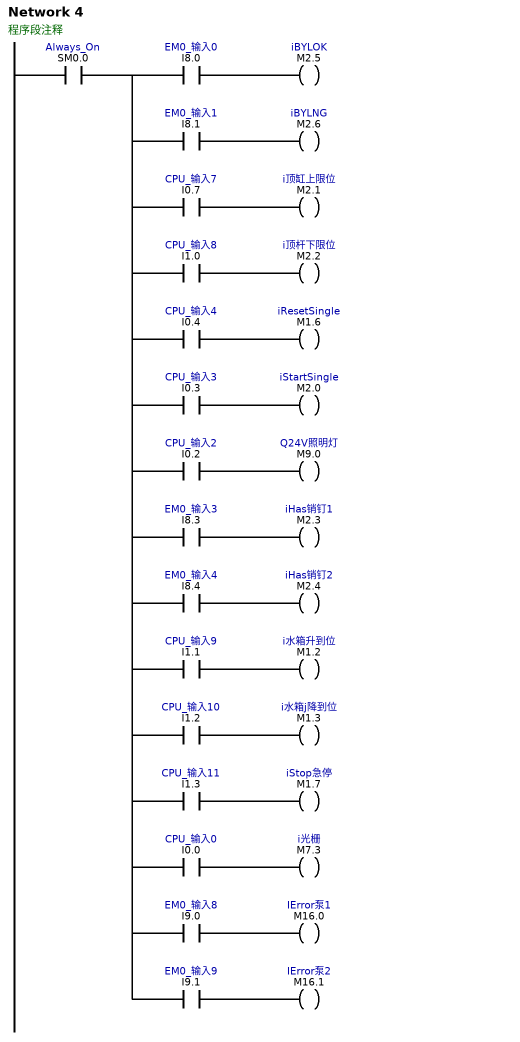
[picture p24: SBR5 networks 4-4]
Network 4
// 程序段注释
LD     Always_On:SM0.0
LPS
A      EM0_输入0:I8.0
=      iBYLOK:M2.5
LRD
A      EM0_输入1:I8.1
=      iBYLNG:M2.6
LRD
A      CPU_输入7:I0.7
=      i顶缸上限位:M2.1
LRD
A      CPU_输入8:I1.0
=      i顶杆下限位:M2.2
LRD
A      CPU_输入4:I0.4
=      iResetSingle:M1.6
LRD
A      CPU_输入3:I0.3
=      iStartSingle:M2.0
LRD
A      CPU_输入2:I0.2
=      Q24V照明灯:M9.0
LRD
A      EM0_输入3:I8.3
=      iHas销钉1:M2.3
LRD
A      EM0_输入4:I8.4
=      iHas销钉2:M2.4
LRD
A      CPU_输入9:I1.1
=      i水箱升到位:M1.2
LRD
A      CPU_输入10:I1.2
=      i水箱j降到位:M1.3
LRD
A      CPU_输入11:I1.3
=      iStop急停:M1.7
LRD
A      CPU_输入0:I0.0
=      i光栅:M7.3
LRD
A      EM0_输入8:I9.0
=      IError泵1:M16.0
LPP
A      EM0_输入9:I9.1
=      IError泵2:M16.1
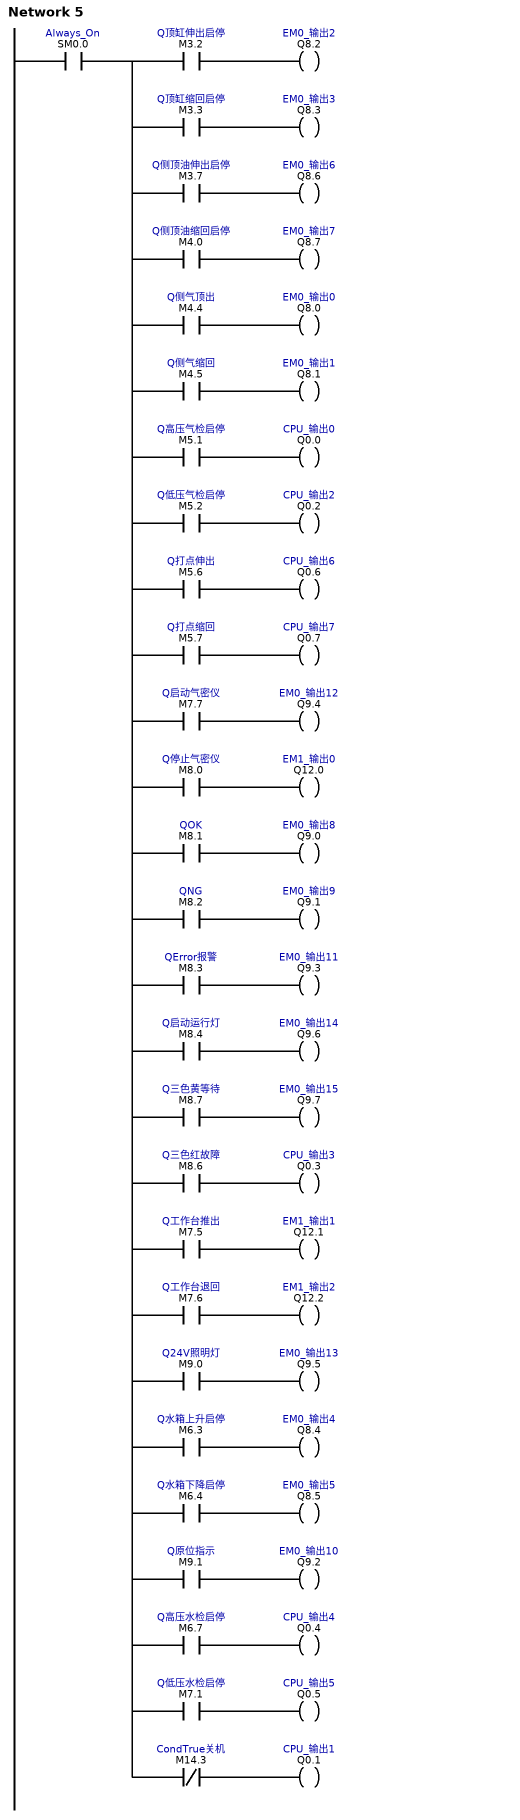
Network 5
LD     Always_On:SM0.0
LPS
A      Q顶缸伸出启停:M3.2
=      EM0_输出2:Q8.2
LRD
A      Q顶缸缩回启停:M3.3
=      EM0_输出3:Q8.3
LRD
A      Q侧顶油伸出启停:M3.7
=      EM0_输出6:Q8.6
LRD
A      Q侧顶油缩回启停:M4.0
=      EM0_输出7:Q8.7
LRD
A      Q侧气顶出:M4.4
=      EM0_输出0:Q8.0
LRD
A      Q侧气缩回:M4.5
=      EM0_输出1:Q8.1
LRD
A      Q高压气检启停:M5.1
=      CPU_输出0:Q0.0
LRD
A      Q低压气检启停:M5.2
=      CPU_输出2:Q0.2
LRD
A      Q打点伸出:M5.6
=      CPU_输出6:Q0.6
LRD
A      Q打点缩回:M5.7
=      CPU_输出7:Q0.7
LRD
A      Q启动气密仪:M7.7
=      EM0_输出12:Q9.4
LRD
A      Q停止气密仪:M8.0
=      EM1_输出0:Q12.0
LRD
A      QOK:M8.1
=      EM0_输出8:Q9.0
LRD
A      QNG:M8.2
=      EM0_输出9:Q9.1
LRD
A      QError报警:M8.3
=      EM0_输出11:Q9.3
LRD
A      Q启动运行灯:M8.4
=      EM0_输出14:Q9.6
LRD
A      Q三色黄等待:M8.7
=      EM0_输出15:Q9.7
LRD
A      Q三色红故障:M8.6
=      CPU_输出3:Q0.3
LRD
A      Q工作台推出:M7.5
=      EM1_输出1:Q12.1
LRD
A      Q工作台退回:M7.6
=      EM1_输出2:Q12.2
LRD
A      Q24V照明灯:M9.0
=      EM0_输出13:Q9.5
LRD
A      Q水箱上升启停:M6.3
=      EM0_输出4:Q8.4
LRD
A      Q水箱下降启停:M6.4
=      EM0_输出5:Q8.5
LRD
A      Q原位指示:M9.1
=      EM0_输出10:Q9.2
LRD
A      Q高压水检启停:M6.7
=      CPU_输出4:Q0.4
LRD
A      Q低压水检启停:M7.1
=      CPU_输出5:Q0.5
LPP
AN     CondTrue关机:M14.3
=      CPU_输出1:Q0.1
END_SUBROUTINE_BLOCK

SUBROUTINE_BLOCK ConverData:SBR6
TITLE=子程序注释
VAR
tmpDint:DINT;	// LD0 
tmpReal:REAL;	// LD4 
END_VAR
BEGIN
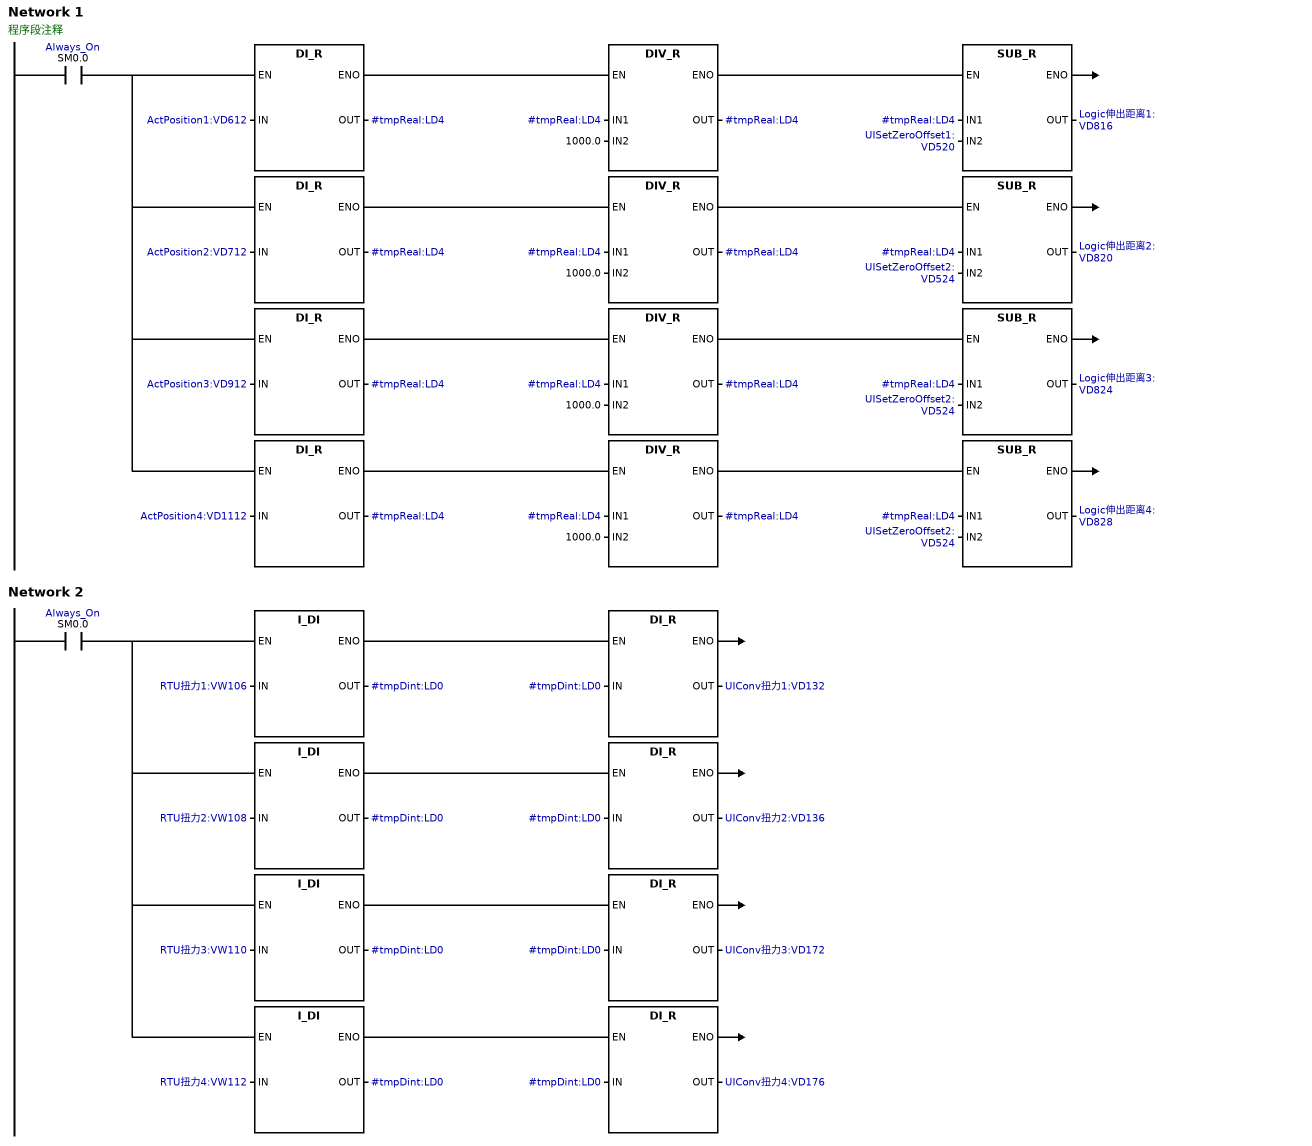
Network 1
// 程序段注释
LD     Always_On:SM0.0
LPS
DTR    ActPosition1:VD612, #tmpReal:LD4
AENO
/R     1000.0, #tmpReal:LD4
AENO
MOVR   #tmpReal:LD4, Logic伸出距离1:VD816
-R     UISetZeroOffset1:VD520, Logic伸出距离1:VD816
LRD
DTR    ActPosition2:VD712, #tmpReal:LD4
AENO
/R     1000.0, #tmpReal:LD4
AENO
MOVR   #tmpReal:LD4, Logic伸出距离2:VD820
-R     UISetZeroOffset2:VD524, Logic伸出距离2:VD820
LRD
DTR    ActPosition3:VD912, #tmpReal:LD4
AENO
/R     1000.0, #tmpReal:LD4
AENO
MOVR   #tmpReal:LD4, Logic伸出距离3:VD824
-R     UISetZeroOffset2:VD524, Logic伸出距离3:VD824
LPP
DTR    ActPosition4:VD1112, #tmpReal:LD4
AENO
/R     1000.0, #tmpReal:LD4
AENO
MOVR   #tmpReal:LD4, Logic伸出距离4:VD828
-R     UISetZeroOffset2:VD524, Logic伸出距离4:VD828
Network 2
LD     Always_On:SM0.0
LPS
ITD    RTU扭力1:VW106, #tmpDint:LD0
AENO
DTR    #tmpDint:LD0, UIConv扭力1:VD132
LRD
ITD    RTU扭力2:VW108, #tmpDint:LD0
AENO
DTR    #tmpDint:LD0, UIConv扭力2:VD136
LRD
ITD    RTU扭力3:VW110, #tmpDint:LD0
AENO
DTR    #tmpDint:LD0, UIConv扭力3:VD172
LPP
ITD    RTU扭力4:VW112, #tmpDint:LD0
AENO
DTR    #tmpDint:LD0, UIConv扭力4:VD176
END_SUBROUTINE_BLOCK

// SBR7: protected block, not included

// SBR8: protected block, not included

SUBROUTINE_BLOCK XinJiePN:SBR9
TITLE=子程序注释
VAR
tmpSpeed:DWORD;	// LD0 
tmpPos1:DINT;	// LD4 
tmpWarning:WORD;	// LW8 
tmpErr:WORD;	// LW10 
tmpDone:BOOL;	// L12.0 
tmpNotJOD:BOOL;	// L12.1 
tmpPos2:DINT;	// LD13 
tmpReal:REAL;	// LD17 
tmpDint:DINT;	// LD21 
tmpPos3:DINT;	// LD25 
tmpPos4:DINT;	// LD29 
END_VAR
BEGIN
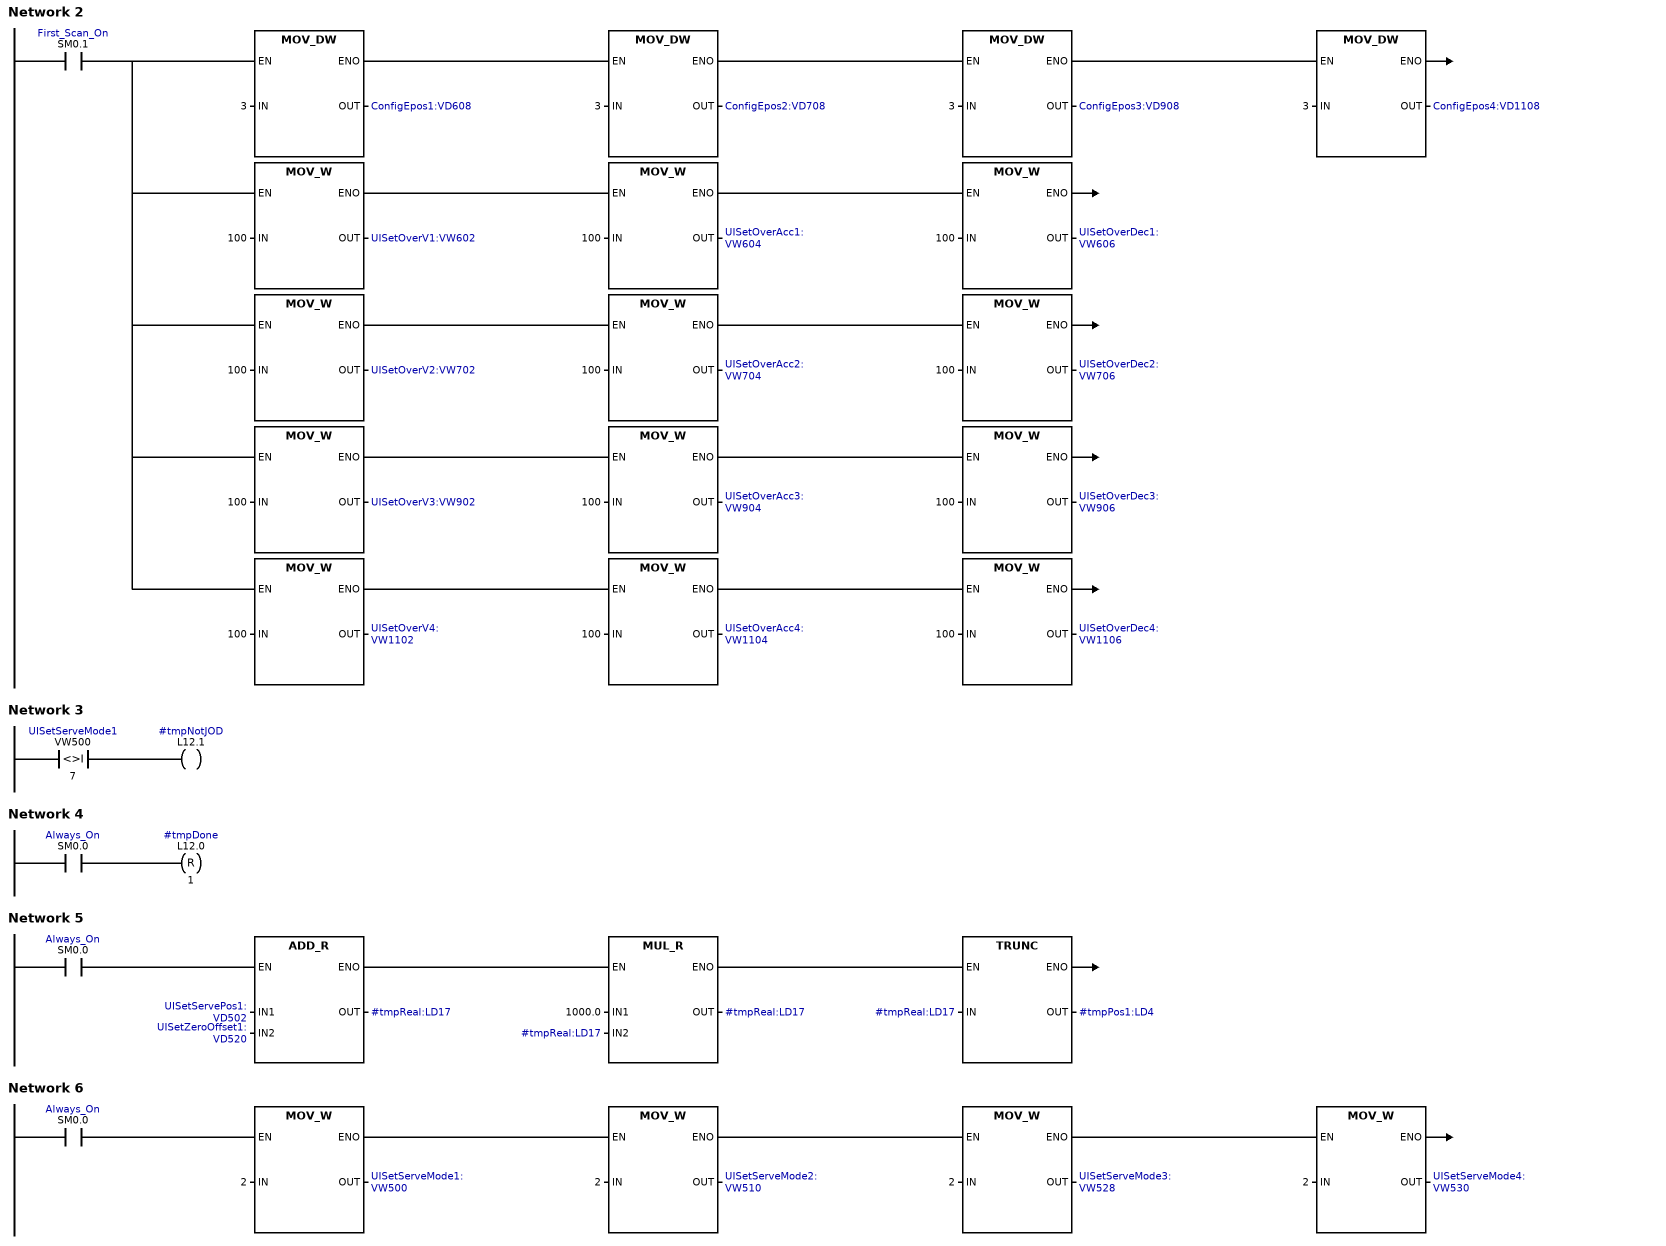
Network 2
LD     First_Scan_On:SM0.1
LPS
MOVD   3, ConfigEpos1:VD608
AENO
MOVD   3, ConfigEpos2:VD708
AENO
MOVD   3, ConfigEpos3:VD908
AENO
MOVD   3, ConfigEpos4:VD1108
LRD
MOVW   100, UISetOverV1:VW602
AENO
MOVW   100, UISetOverAcc1:VW604
AENO
MOVW   100, UISetOverDec1:VW606
LRD
MOVW   100, UISetOverV2:VW702
AENO
MOVW   100, UISetOverAcc2:VW704
AENO
MOVW   100, UISetOverDec2:VW706
LRD
MOVW   100, UISetOverV3:VW902
AENO
MOVW   100, UISetOverAcc3:VW904
AENO
MOVW   100, UISetOverDec3:VW906
LPP
MOVW   100, UISetOverV4:VW1102
AENO
MOVW   100, UISetOverAcc4:VW1104
AENO
MOVW   100, UISetOverDec4:VW1106
Network 3
LDW<>  UISetServeMode1:VW500, 7
=      #tmpNotJOD:L12.1
Network 4
LD     Always_On:SM0.0
R      #tmpDone:L12.0, 1
Network 5
LD     Always_On:SM0.0
MOVR   UISetServePos1:VD502, #tmpReal:LD17
AENO
+R     UISetZeroOffset1:VD520, #tmpReal:LD17
AENO
*R     1000.0, #tmpReal:LD17
AENO
TRUNC  #tmpReal:LD17, #tmpPos1:LD4
Network 6
LD     Always_On:SM0.0
MOVW   2, UISetServeMode1:VW500
AENO
MOVW   2, UISetServeMode2:VW510
AENO
MOVW   2, UISetServeMode3:VW528
AENO
MOVW   2, UISetServeMode4:VW530
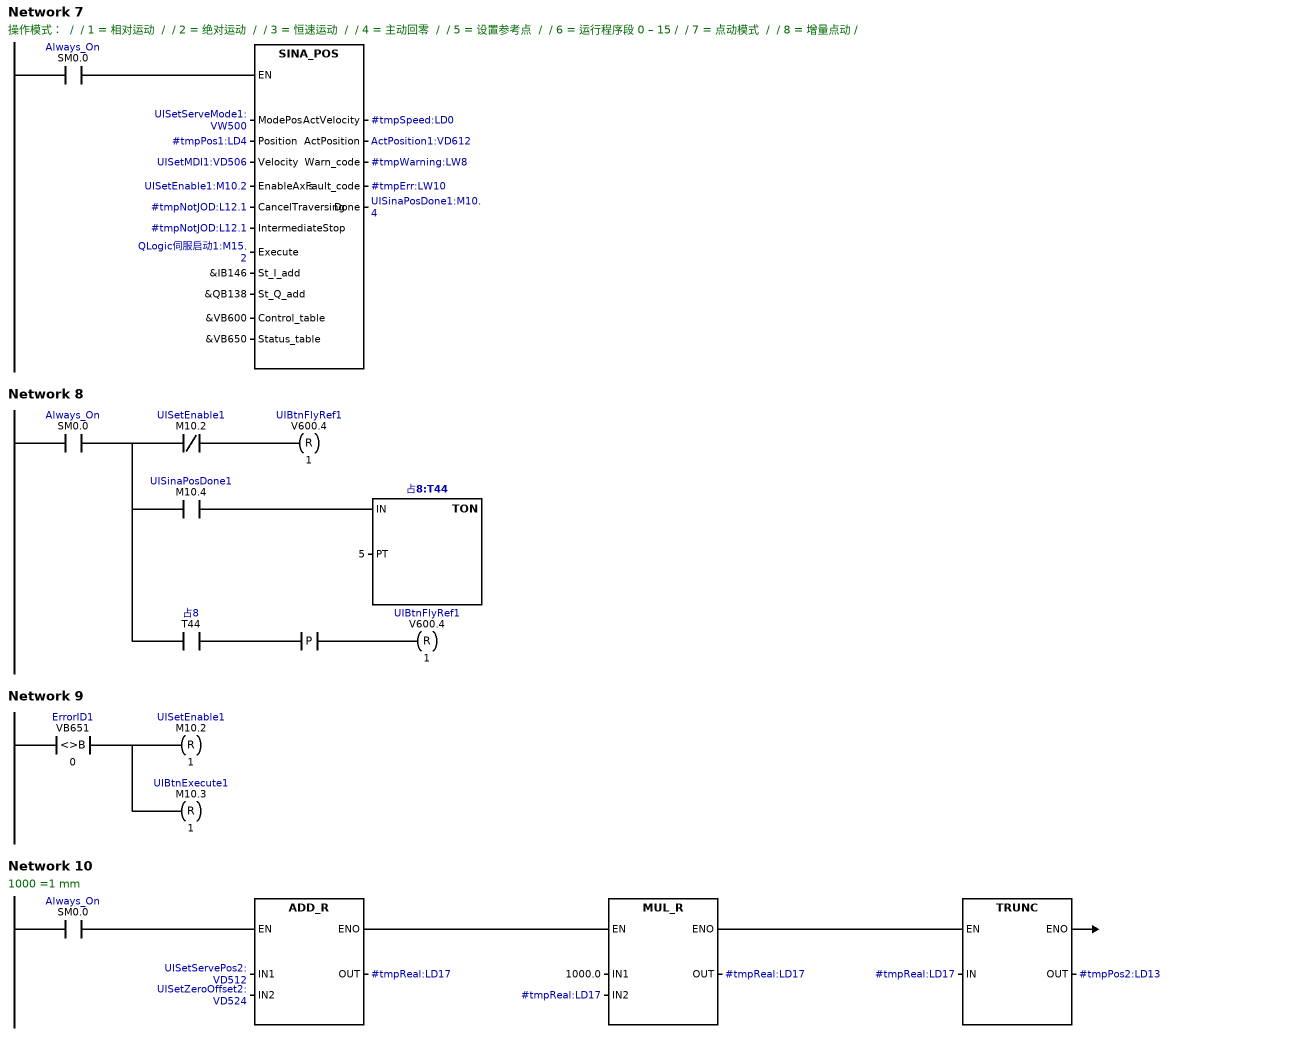
Network 7
// 操作模式： 
// 
// 1 = 相对运动 
// 
// 2 = 绝对运动 
// 
// 3 = 恒速运动 
// 
// 4 = 主动回零 
// 
// 5 = 设置参考点 
// 
// 6 = 运行程序段 0 – 15
// 
// 7 = 点动模式 
// 
// 8 = 增量点动
// 
LD     Always_On:SM0.0
CALL   SINA_POS:SBR8, UISetServeMode1:VW500, #tmpPos1:LD4, UISetMDI1:VD506, UISetEnable1:M10.2, #tmpNotJOD:L12.1, #tmpNotJOD:L12.1, QLogic伺服启动1:M15.2, &IB146, &QB138, &VB600, &VB650, #tmpSpeed:LD0, ActPosition1:VD612, #tmpWarning:LW8, #tmpErr:LW10, UISinaPosDone1:M10.4
Network 8
LD     Always_On:SM0.0
LPS
AN     UISetEnable1:M10.2
R      UIBtnFlyRef1:V600.4, 1
LRD
A      UISinaPosDone1:M10.4
TON    占8:T44, 5
LPP
A      占8:T44
EU
R      UIBtnFlyRef1:V600.4, 1
Network 9
LDB<>  ErrorID1:VB651, 0
R      UISetEnable1:M10.2, 1
R      UIBtnExecute1:M10.3, 1
Network 10
//  1000 =1 mm
LD     Always_On:SM0.0
MOVR   UISetServePos2:VD512, #tmpReal:LD17
AENO
+R     UISetZeroOffset2:VD524, #tmpReal:LD17
AENO
*R     1000.0, #tmpReal:LD17
AENO
TRUNC  #tmpReal:LD17, #tmpPos2:LD13
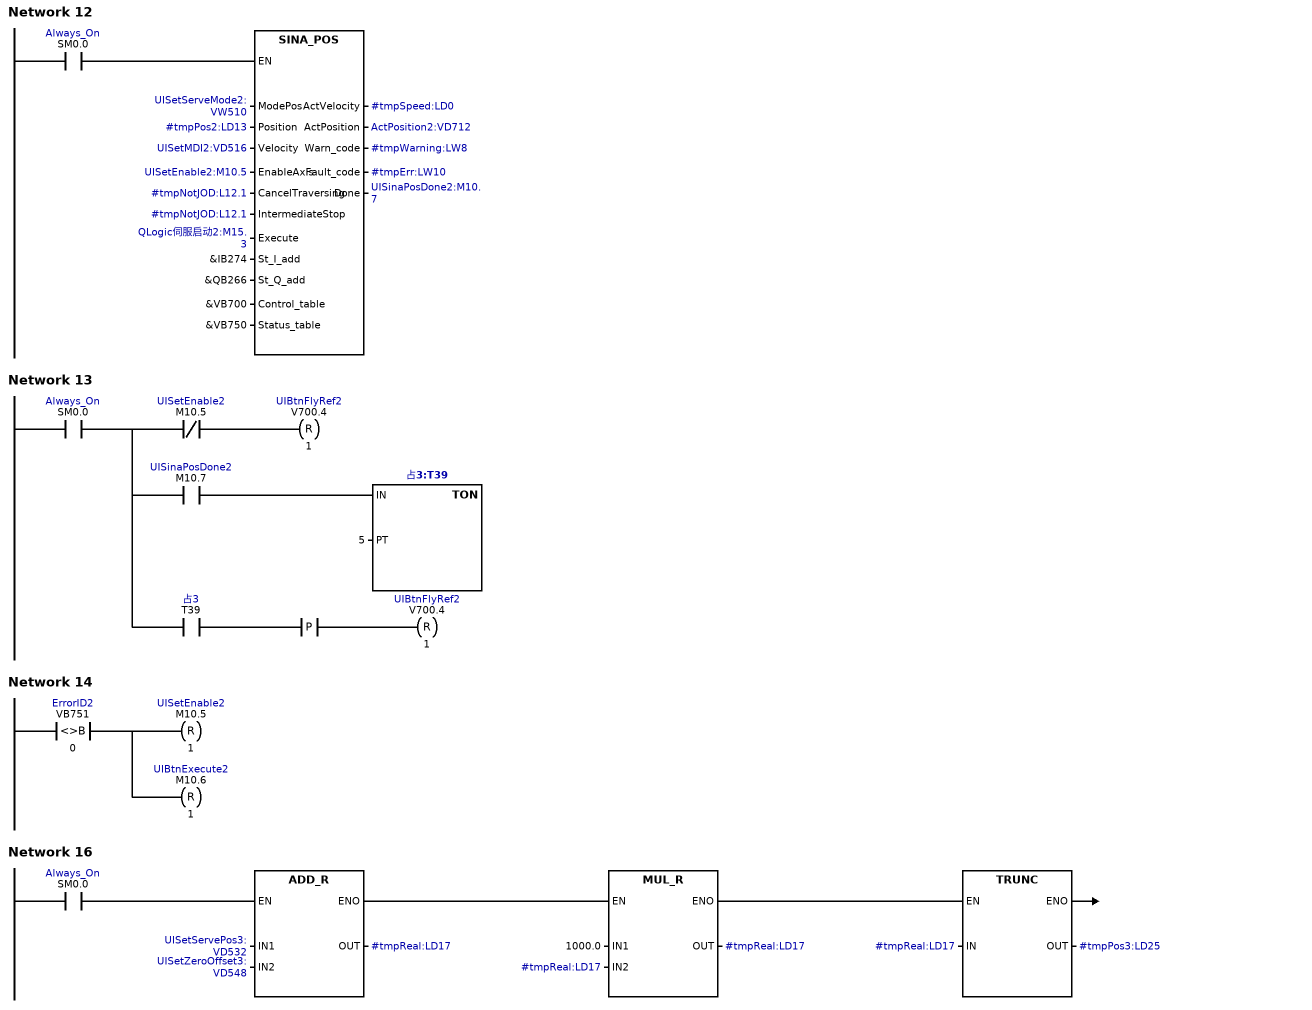
Network 12
LD     Always_On:SM0.0
CALL   SINA_POS:SBR8, UISetServeMode2:VW510, #tmpPos2:LD13, UISetMDI2:VD516, UISetEnable2:M10.5, #tmpNotJOD:L12.1, #tmpNotJOD:L12.1, QLogic伺服启动2:M15.3, &IB274, &QB266, &VB700, &VB750, #tmpSpeed:LD0, ActPosition2:VD712, #tmpWarning:LW8, #tmpErr:LW10, UISinaPosDone2:M10.7
Network 13
LD     Always_On:SM0.0
LPS
AN     UISetEnable2:M10.5
R      UIBtnFlyRef2:V700.4, 1
LRD
A      UISinaPosDone2:M10.7
TON    占3:T39, 5
LPP
A      占3:T39
EU
R      UIBtnFlyRef2:V700.4, 1
Network 14
LDB<>  ErrorID2:VB751, 0
R      UISetEnable2:M10.5, 1
R      UIBtnExecute2:M10.6, 1
Network 16
LD     Always_On:SM0.0
MOVR   UISetServePos3:VD532, #tmpReal:LD17
AENO
+R     UISetZeroOffset3:VD548, #tmpReal:LD17
AENO
*R     1000.0, #tmpReal:LD17
AENO
TRUNC  #tmpReal:LD17, #tmpPos3:LD25
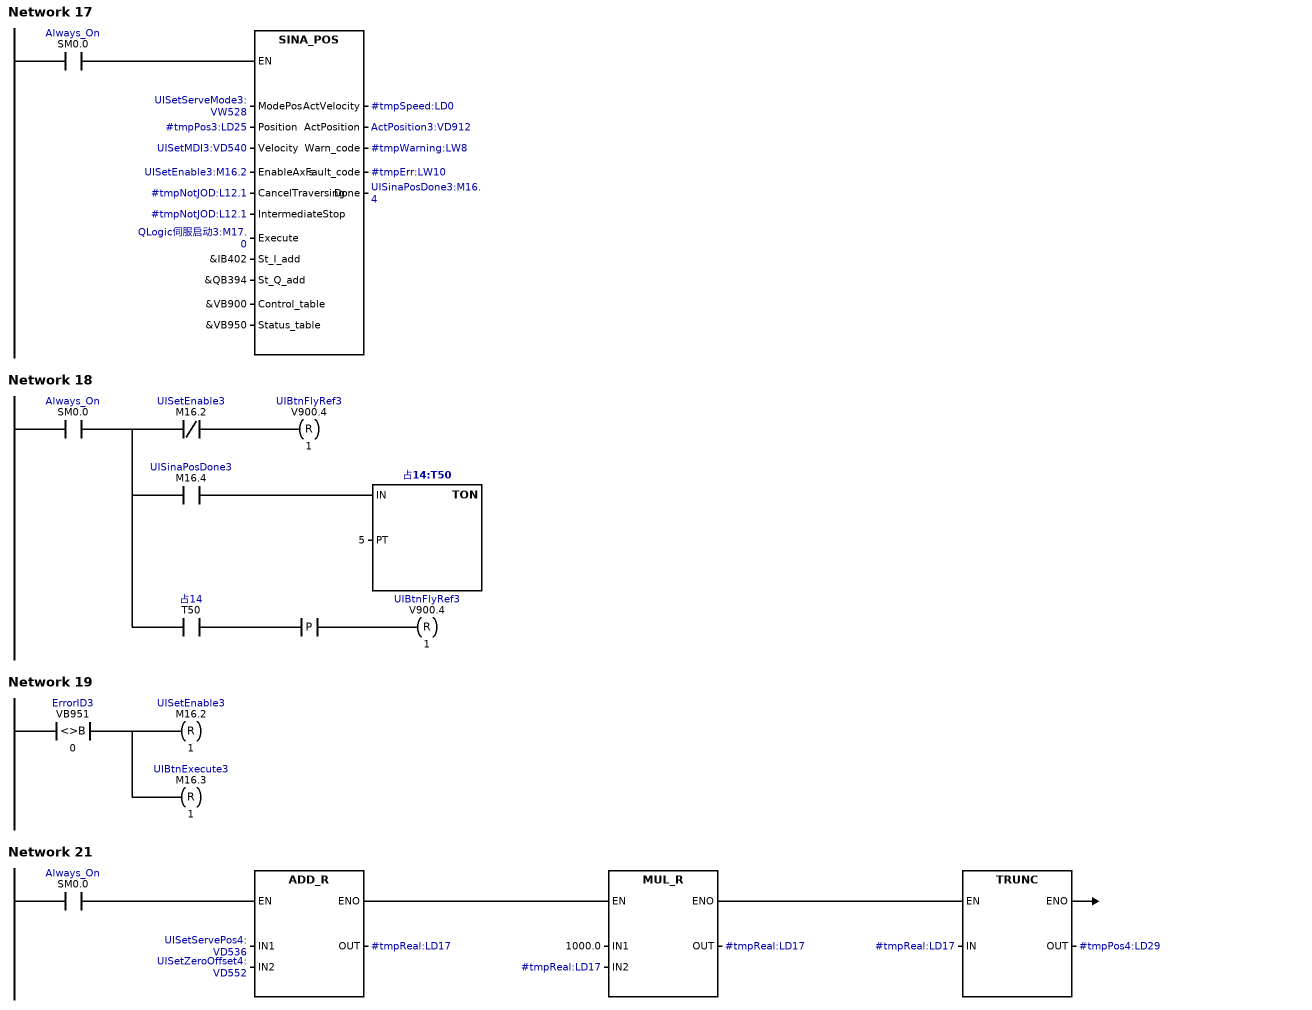
Network 17
LD     Always_On:SM0.0
CALL   SINA_POS:SBR8, UISetServeMode3:VW528, #tmpPos3:LD25, UISetMDI3:VD540, UISetEnable3:M16.2, #tmpNotJOD:L12.1, #tmpNotJOD:L12.1, QLogic伺服启动3:M17.0, &IB402, &QB394, &VB900, &VB950, #tmpSpeed:LD0, ActPosition3:VD912, #tmpWarning:LW8, #tmpErr:LW10, UISinaPosDone3:M16.4
Network 18
LD     Always_On:SM0.0
LPS
AN     UISetEnable3:M16.2
R      UIBtnFlyRef3:V900.4, 1
LRD
A      UISinaPosDone3:M16.4
TON    占14:T50, 5
LPP
A      占14:T50
EU
R      UIBtnFlyRef3:V900.4, 1
Network 19
LDB<>  ErrorID3:VB951, 0
R      UISetEnable3:M16.2, 1
R      UIBtnExecute3:M16.3, 1
Network 21
LD     Always_On:SM0.0
MOVR   UISetServePos4:VD536, #tmpReal:LD17
AENO
+R     UISetZeroOffset4:VD552, #tmpReal:LD17
AENO
*R     1000.0, #tmpReal:LD17
AENO
TRUNC  #tmpReal:LD17, #tmpPos4:LD29
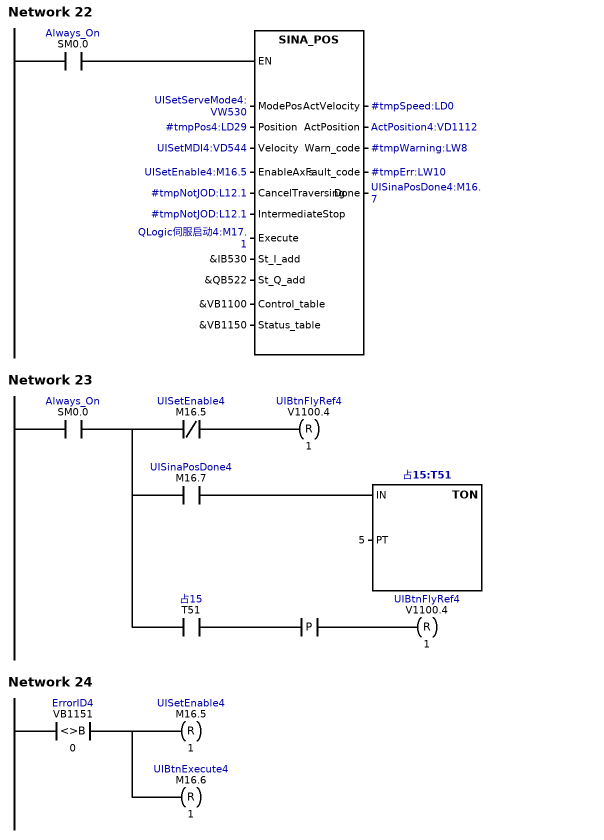
Network 22
LD     Always_On:SM0.0
CALL   SINA_POS:SBR8, UISetServeMode4:VW530, #tmpPos4:LD29, UISetMDI4:VD544, UISetEnable4:M16.5, #tmpNotJOD:L12.1, #tmpNotJOD:L12.1, QLogic伺服启动4:M17.1, &IB530, &QB522, &VB1100, &VB1150, #tmpSpeed:LD0, ActPosition4:VD1112, #tmpWarning:LW8, #tmpErr:LW10, UISinaPosDone4:M16.7
Network 23
LD     Always_On:SM0.0
LPS
AN     UISetEnable4:M16.5
R      UIBtnFlyRef4:V1100.4, 1
LRD
A      UISinaPosDone4:M16.7
TON    占15:T51, 5
LPP
A      占15:T51
EU
R      UIBtnFlyRef4:V1100.4, 1
Network 24
LDB<>  ErrorID4:VB1151, 0
R      UISetEnable4:M16.5, 1
R      UIBtnExecute4:M16.6, 1
END_SUBROUTINE_BLOCK

// SBR10: protected block, not included

// SBR11: protected block, not included

// SBR12: protected block, not included
